	                //VID
	                #iq_UDT_MessageData.XrayRegistrationInfo.VID := CONCAT(IN1 := BYTE_TO_CHAR(#s_UDT_FifoMessage.Bytes[8]),
	                                                                       IN2 := BYTE_TO_CHAR(#s_UDT_FifoMessage.Bytes[9]),
	                                                                       IN3 := BYTE_TO_CHAR(#s_UDT_FifoMessage.Bytes[10]),
	                                                                       IN4 := BYTE_TO_CHAR(#s_UDT_FifoMessage.Bytes[11]),
	                                                                       IN5 := BYTE_TO_CHAR(#s_UDT_FifoMessage.Bytes[12]),
	                                                                       IN6 := BYTE_TO_CHAR(#s_UDT_FifoMessage.Bytes[13]),
	                                                                       IN7 := BYTE_TO_CHAR(#s_UDT_FifoMessage.Bytes[14]),
	                                                                       IN8 := BYTE_TO_CHAR(#s_UDT_FifoMessage.Bytes[15]),
	                                                                       IN9 := BYTE_TO_CHAR(#s_UDT_FifoMessage.Bytes[16]),
	                                                                       IN10 := BYTE_TO_CHAR(#s_UDT_FifoMessage.Bytes[17]),
	                                                                       IN11 := BYTE_TO_CHAR(#s_UDT_FifoMessage.Bytes[18]),
	                                                                       IN12 := BYTE_TO_CHAR(#s_UDT_FifoMessage.Bytes[19]),
	                                                                       IN13 := BYTE_TO_CHAR(#s_UDT_FifoMessage.Bytes[20]),
	                                                                       IN14 := BYTE_TO_CHAR(#s_UDT_FifoMessage.Bytes[21]),
	                                                                       IN15 := BYTE_TO_CHAR(#s_UDT_FifoMessage.Bytes[22]),
	                                                                       IN16 := BYTE_TO_CHAR(#s_UDT_FifoMessage.Bytes[23]));

	                //Piece ID
	                #iq_UDT_MessageData.XrayRegistrationInfo.PieceID := CONCAT(IN1 := BYTE_TO_CHAR(#s_UDT_FifoMessage.Bytes[24]),
	                                                                           IN2 := BYTE_TO_CHAR(#s_UDT_FifoMessage.Bytes[25]),
	                                                                           IN3 := BYTE_TO_CHAR(#s_UDT_FifoMessage.Bytes[26]),
	                                                                           IN4 := BYTE_TO_CHAR(#s_UDT_FifoMessage.Bytes[27]),
	                                                                           IN5 := BYTE_TO_CHAR(#s_UDT_FifoMessage.Bytes[28]),
	                                                                           IN6 := BYTE_TO_CHAR(#s_UDT_FifoMessage.Bytes[29]),
	                                                                           IN7 := BYTE_TO_CHAR(#s_UDT_FifoMessage.Bytes[30]),
	                                                                           IN8 := BYTE_TO_CHAR(#s_UDT_FifoMessage.Bytes[31]),
	                                                                           IN9 := BYTE_TO_CHAR(#s_UDT_FifoMessage.Bytes[32]),
	                                                                           IN10 := BYTE_TO_CHAR(#s_UDT_FifoMessage.Bytes[33]),
	                                                                           IN11 := BYTE_TO_CHAR(#s_UDT_FifoMessage.Bytes[34]),
	                                                                           IN12 := BYTE_TO_CHAR(#s_UDT_FifoMessage.Bytes[35]),
	                                                                           IN13 := BYTE_TO_CHAR(#s_UDT_FifoMessage.Bytes[36]),
	                                                                           IN14 := BYTE_TO_CHAR(#s_UDT_FifoMessage.Bytes[37]),
	                                                                           IN15 := BYTE_TO_CHAR(#s_UDT_FifoMessage.Bytes[38]),
	                                                                           IN16 := BYTE_TO_CHAR(#s_UDT_FifoMessage.Bytes[39]),
	                                                                           IN17 := BYTE_TO_CHAR(#s_UDT_FifoMessage.Bytes[40]),
	                                                                           IN18 := BYTE_TO_CHAR(#s_UDT_FifoMessage.Bytes[41]),
	                                                                           IN19 := BYTE_TO_CHAR(#s_UDT_FifoMessage.Bytes[42]),
	                                                                           IN20 := BYTE_TO_CHAR(#s_UDT_FifoMessage.Bytes[43]),
	                                                                           IN21 := BYTE_TO_CHAR(#s_UDT_FifoMessage.Bytes[44]),
	                                                                           IN22 := BYTE_TO_CHAR(#s_UDT_FifoMessage.Bytes[45]),
	                                                                           IN23 := BYTE_TO_CHAR(#s_UDT_FifoMessage.Bytes[46]),
	                                                                           IN24 := BYTE_TO_CHAR(#s_UDT_FifoMessage.Bytes[47]),
	                                                                           IN25 := BYTE_TO_CHAR(#s_UDT_FifoMessage.Bytes[48]),
	                                                                           IN26 := BYTE_TO_CHAR(#s_UDT_FifoMessage.Bytes[49]),
	                                                                           IN27 := BYTE_TO_CHAR(#s_UDT_FifoMessage.Bytes[50]),
	                                                                           IN28 := BYTE_TO_CHAR(#s_UDT_FifoMessage.Bytes[51]),
	                                                                           IN29 := BYTE_TO_CHAR(#s_UDT_FifoMessage.Bytes[52]),
	                                                                           IN30 := BYTE_TO_CHAR(#s_UDT_FifoMessage.Bytes[53]),
	                                                                           IN31 := BYTE_TO_CHAR(#s_UDT_FifoMessage.Bytes[54]),
	                                                                           IN32 := BYTE_TO_CHAR(#s_UDT_FifoMessage.Bytes[55]));

	                #iq_UDT_MessageData.XrayRegistrationInfo.PieceID := CONCAT(IN1 := #iq_UDT_MessageData.XrayRegistrationInfo.PieceID,
	                                                                           IN2 := BYTE_TO_CHAR(#s_UDT_FifoMessage.Bytes[56]),
	                                                                           IN3 := BYTE_TO_CHAR(#s_UDT_FifoMessage.Bytes[57]),
	                                                                           IN4 := BYTE_TO_CHAR(#s_UDT_FifoMessage.Bytes[58]),
	                                                                           IN5 := BYTE_TO_CHAR(#s_UDT_FifoMessage.Bytes[59]),
	                                                                           IN6 := BYTE_TO_CHAR(#s_UDT_FifoMessage.Bytes[60]),
	                                                                           IN7 := BYTE_TO_CHAR(#s_UDT_FifoMessage.Bytes[61]),
	                                                                           IN8 := BYTE_TO_CHAR(#s_UDT_FifoMessage.Bytes[62]),
	                                                                           IN9 := BYTE_TO_CHAR(#s_UDT_FifoMessage.Bytes[63]));


	                //Routing Code - Changed on version 1.1
	                #ts_RoutingCode := DELETE(IN := UDINT_TO_STRING(BYTE_TO_UINT(#s_UDT_FifoMessage.Bytes[64])), L := 1, P := 1);
	                #ts_RoutingCode := CONCAT(IN1 := '0', IN2 := #ts_RoutingCode);      //add leading zero ( 1 -> 01 , 22 -> 022)
	                #ts_RoutingCode := RIGHT(IN := #ts_RoutingCode, L := 2);            //take always last two characters  ( 01-> 01 , 022-> 22)
	                #iq_UDT_MessageData.XrayRegistrationInfo.RoutingCode := #ts_RoutingCode;

	                //Only statistics
	                #ss_CounterRecivedMessage.XrayRegistrationInfo += 1;

	            ELSE

	                #tx_InvalidMessageID := TRUE;

	                //Only statistics
	                #ss_CounterRecivedMessage.InvalidMessageID += 1;

	        END_CASE;

	    END_IF;

	END_REGION

	REGION 3 – Heartbeat monitoring

	    //HB timeout validation.
	    #ss_Status.InvalidTimeout := #iudi_HeartbeatTimeout <= 0;

	    //HB monitoring if timeout correct.
	    IF NOT #ss_Status.InvalidTimeout
	    THEN
	        #s_R_TRIG_Connected(CLK := #ix_Connected);

	        // Heartbeat timeout monitoring.
	        #s_FB_TimerHeartbeatCheck(iudi_OnDelayTime := 0,
	                                  iudi_OffDelayTime := #iudi_HeartbeatTimeout,
	                                  ix_SignalToDelay := #sx_Heartbeat OR #s_R_TRIG_Connected.Q,
	                                  qx_DelayedSignal => #sx_HeartbeatOK);

	        #sx_Heartbeat := FALSE;
	        #s_F_TRIG_HeartbeatNotOk(CLK := #sx_HeartbeatOK);

	        IF #s_F_TRIG_HeartbeatNotOk.Q
	            AND "DB_Memory".AlwaysFalse
	        THEN
	            // Re-establish conncect with partner and increment the number of communication lost.
	            #iqx_Reconnect := TRUE;
	            #iq_UDT_Statistics.HeartbeatNotObserved += 1;
	        END_IF;
	    END_IF;

	END_REGION

	REGION 4 – Statistics update

	    // Error statistics update required.
	    IF #tx_InvalidHeader
	        OR #tx_InvalidMessageID
	        OR #tx_BadMessage
	    THEN
	        // Invalid message received counter incrementation.
	        #iq_UDT_Statistics.InvalidMessage += 1;

	        // Maximum number of bad messages array.
	        #ti_BadMessageSize := "FC_GetNrOfArrayEl"(#ss_Status.BadMessage);

	        // Writing invalid message in a bad message array.
	        IF #si_RingBufferNumber >= #ti_BadMessageSize
	        THEN
	            #si_RingBufferNumber := 1;
	        END_IF;

	        #ti_NumberOfMessageBytes := "FC_GetNrOfArrayEl"(iv_Array := #s_UDT_FifoMessage.Bytes);

	        MOVE_BLK(IN := #s_UDT_FifoMessage.Bytes[0],
	                 COUNT := INT_TO_UINT(#ti_NumberOfMessageBytes) - 1,
	                 OUT => #ss_Status.BadMessage[#si_RingBufferNumber].Bytes[0]);

	        #si_RingBufferNumber += 1;
	    END_IF;

	    //Resetting statistics.
	    IF #ix_ResetData
	    THEN
	        #iq_UDT_Statistics.InvalidMessage := 0;
	        #iq_UDT_Statistics.HeartbeatNotObserved := 0;
	    END_IF;

	END_REGION

	REGION 5 – Status

	    // Collective error output.
	    #qx_Error :=
	    #ss_Status.FIFOReceiveError
	    OR #ss_Status.InvalidTimeout;

	    // Collective warning output.
	    #qx_Warning :=
	    #ss_Status.FIFOReceiveWarning;

	END_REGION




END_FUNCTION_BLOCK

